Staubli VAL3: TP1_Paolo.pjx

--- TP1_Paolo.pjx ---
Parameters version=s7.5 stackSize=5000 millimeterUnit=true
Program file=picketplace.pgx
Program file=start.pgx
Program file=stop.pgx
Data file=TP1_Paolo.dtx

--- TP1_Paolo.dtx ---
frame fTable = {x=544.793496, y=2.880447, z=-170.95, rx=-179.999977, ry=-0.0003, rz=0.000308, fatherId=world[0]}
jointRx j0
jointRx jDepart = {j1=-7.215316, j2=54.432296, j3=135.763663, j4=-6.983157, j5=-101.065649, j6=-91.233508}
mdesc mPriseDepose = {vel=5}
mdesc mRapide100joint = {vel=25}
pointRx pDepose[2]
  [0] = {x=80.895535, y=164.405443, z=205.485609, rx=20.949006, ry=91.010648, rz=69.047818, fatherId=fTable[0]}
  [1] = {x=83.817549, y=-298.865741, z=205.487219, rx=20.949006, ry=91.010648, rz=69.047818, fatherId=fTable[0]}
pointRx pPrise = {x=81.971792, y=-6.229802, z=205.486202, rx=20.949006, ry=91.010648, rz=69.047818, fatherId=fTable[0]}
sio sData = {link=Socket\staubli_server}
tool tPince = {x=-1.667681, y=-1.981137, z=74.877299, rx=0, ry=0, rz=0, fatherId=flange[0], ioLink=valve1}
trsf trApproZ = {z=-50}

--- start.pgx ---
program start()
  local num l_ncouleur_bout
begin

  //  sioCtrl(sData, "port", 8500)
  //  sioCtrl(sData, "clients", 1)
  //  //CCaractère de fin de line : Line Feed
  //  sioCtrl(sData, "endOfString", 13)

  //  logMsg("------------ Sio Initialise")

  //  logMsg("  dataAcquisition start")
  //  do

  //    nb=0
  //    i=0
  //    while(nb<32)
  //      nb=sioGet(sData, l_nByteIn[i])

  //      if(nb>0)
  //        i=i+nb
  //      else
  //        // Erreur de communication
  //        return
  //      endIf
  //      logMsg("Recuperation du buffer...")
  //    endWhile
  //    logMsg("Buffer récupéré.")



  l_ncouleur_bout=1

  call picketplace(l_ncouleur_bout)


  l_ncouleur_bout=0
  call picketplace(l_ncouleur_bout)
  waitEndMove()

end

--- picketplace.pgx ---
program picketplace(num x_nCouleurbout (dimensions=1))
begin
  // 1er Mouvement sur un Joint
  movej(jDepart,tPince,mRapide100joint)



  movej(appro(pPrise[0],trApproZ),tPince,mRapide100joint)

  // Ouvrir la Pince
  open(tPince)
  // Aller Lentement au Point de Prise
  movel(pPrise[0],tPince,mPriseDepose)
  // Fermer la Pince
  close(tPince)

  // Aller Lentement au Point d'Approche Prise (Dégagement)
  movel(appro(pPrise[0],trApproZ),tPince,mPriseDepose)


  // 3 Mouvements pour la Depose de la Bouteille
  // Aller Rapidement au Point d'Approche Depose selon la couleur de la bouteille
  movej(appro(pDepose[x_nCouleurbout],trApproZ),tPince,mRapide100joint)

  // Aller Lentement au Point de Depose
  movel(pDepose[x_nCouleurbout],tPince,mPriseDepose)

  open(tPince)

  // Aller Lentement au Point d'Approche Depose (Dégagement)
  movel(appro(pDepose[x_nCouleurbout],trApproZ),tPince,mPriseDepose)


  // Dernier Mouvement sur un Joint
  movej(jDepart,tPince,mRapide100joint)

end
